Fanuc KAREL source: ko00029.KL

-- PROVISIONAL review KL for V770-1; original PC SHA256 26894785d711d9f0ecf6ed6414d30601cc9dba9c1feefac2d7a5d19f9a56b8f7
-- Incomplete behavior may be omitted. Consult companion uncertainty JSON. Do not deploy.
PROGRAM KO00029
%NOLOCKGROUP
-- UNRESOLVED_DECL P1 type=000199
-- UNRESOLVED_DECL P2 type=000199
-- UNRESOLVED_DECL P3 type=000199
-- UNRESOLVED_DECL P4 type=000199
-- UNRESOLVED_DECL OUT type=000101
BEGIN
  -- UNRESOLVED_PC offsets 5-80; opcodes 27,27,49,7E,AD,27,49,7E,AD,27,49,7E,AD,27,49,7E,AD,76,7E,4A
  -- UNRESOLVED_PC offsets 85-89; opcodes 7F
END KO00029
